// Mitsubishi GX Works2 project: 실린더제어ABBA   PLC: Q02/Q02H

PROGRAM MAIN
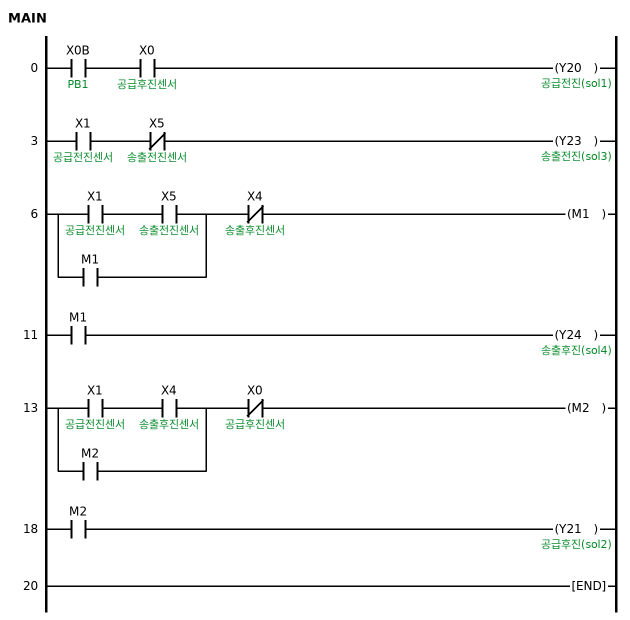
0     LD      X0B  ; PB1
      AND     X0  ; 공급후진센서
      OUT     Y20  ; 공급전진(sol1)
3     LD      X1  ; 공급전진센서
      ANI     X5  ; 송출전진센서
      OUT     Y23  ; 송출전진(sol3)
6     LD      X1  ; 공급전진센서
      AND     X5  ; 송출전진센서
      OR      M1
      ANI     X4  ; 송출후진센서
      OUT     M1
11    LD      M1
      OUT     Y24  ; 송출후진(sol4)
13    LD      X1  ; 공급전진센서
      AND     X4  ; 송출후진센서
      OR      M2
      ANI     X0  ; 공급후진센서
      OUT     M2
18    LD      M2
      OUT     Y21  ; 공급후진(sol2)
20    END
END_PROGRAM

// device comments not shown above
X0C  ; PB2
X0D  ; PB3
